{attribute 'linkalways'} 
{attribute 'no_explicit_call' := 'This FB is a CLASS and must be accessed using methods or properties'}
{attribute 'enable_dynamic_creation'}
FUNCTION_BLOCK FINAL SUB_DINT EXTENDS Node
VAR
	in1 : _DINT(0);
	in2 : _DINT(0);
	out : _DINT(0);
END_VAR

METHOD PUBLIC Clone : I_Node
VAR
	pNode : POINTER TO SUB_DINT;
END_VAR
pNode := __NEW(SUB_DINT);
Clone := pNode^;
END_METHOD

METHOD FB_init : BOOL
VAR_INPUT
	bInitRetains : BOOL; // if TRUE, the retain variables are initialized (warm start / cold start)
	bInCopyCode : BOOL;  // if TRUE, the instance afterwards gets moved into the copy code (online change)
END_VAR
AddInput('in1',THIS^.in1);
AddInput('in2',THIS^.in2);
AddOutput('out', THIS^.out);
END_METHOD

METHOD PROTECTED OnExecute
VAR
END_VAR
out.Value := in1.Value - in2.Value;
END_METHOD

END_FUNCTION_BLOCK

(* stored: Version 1.1.0.1, ProductVersion 3.1.4024.15
   POU SUB_DINT: Id {6402f82b-d876-4956-8a28-af1d834acbe6}, SpecialFunc None
   Folder Constructor: Id {26416eb8-9786-4462-a013-d8b302b7475a}
   Method Clone: Id {f4ea3209-2b8f-4941-b503-7130d5c7bcb0}
   Method FB_init: Id {0891ca71-a3da-4da9-ac68-a0b574abbcb5}
   Method OnExecute: Id {bebaea51-32b8-4c77-93fa-d11bdfe49a82} *)
